// TIA Portal V20 export
// export: Created 2026-09-14T11:29:01.1145551Z, ExportSetting None, DisplayName Totally Integrated Automation Portal, DisplayVersion V20, DisplayName TIA Portal Openness, DisplayVersion V20, DisplayName TIA Portal Version Control Interface, DisplayVersion V20, DisplayName STEP 7 Professional, DisplayVersion V20, DisplayName STEP 7 Safety, DisplayVersion V20, DisplayName WinCC Basic/Comfort/Advanced, DisplayVersion V20, DisplayName WinCC Unified, DisplayVersion V20
TYPE "LMQTT_typeSubscribeData"
   STRUCT
      subscribeToTopic : Bool;   // When true, subscribes to the topic indicated by "subscriptionTopic"
      unsubscribeFromTopic : Bool;   // When true, unsubscribes from the "subscriptionTopic"
      subscriptionTopic : WString[250];   // Topic name to subscribe to or unsubscribe off
      subscriptionQoS : Int;   // Defines the QoS level for the MQTT message at the subscriber side. 0 and 1 allowed
   END_STRUCT;
END_TYPE
